INTERFACE I_AnalogCommandable

METHOD SetValue : E_RpcMethodResponse
VAR_INPUT
    rValue : REAL;
    eRequester : E_Requester := E_Requester.PROG;
END_VAR
END_METHOD

END_INTERFACE

(* stored: Version 1.1.0.1, ProductVersion 3.1.4026.12
   Itf I_AnalogCommandable: Id {c0000005-0000-0000-0000-000000000001}
   Method SetValue: Id {c0000005-0000-0000-1000-000000000001} *)
